TYPE "PnDiag_Alr"
VERSION : 0.1
// Block: PnDiag_Alr
   STRUCT
      Error : Bool;
      Module_Error : Bool;
   END_STRUCT;

END_TYPE
